(*

.. <legal notes>

legal notes
=================
| SPDX-FileCopyrightText: © 2026 Oleksandr Tiutyk <trofimich@gmail.com>
| SPDX-License-Identifier: LGPL-3.0-only
| For details check: LGPL-3.0-only_

.. _LGPL-3.0-only: https://www.gnu.org/licenses/lgpl-3.0.en.html

.. </legal notes>

*)

FUNCTION_BLOCK ABSTRACT LeafAutomationComponent EXTENDS AutomationComponent IMPLEMENTS IChildAutomationComponent
VAR
	{attribute 'hide'} 
	_Parent : IParentAutomationComponent;
END_VAR

METHOD FINAL BubbleEvent
VAR_INPUT
	event : TOF_Core.IEvent;
END_VAR
VAR
	stopPropagation : BOOL;
	
	parentAsBubbleEventDispatcher : TOF_Core.IBubbleEventDispatcher;
END_VAR
OnEventReceived(event := event, stopPropagation => stopPropagation);

IF stopPropagation THEN
	RETURN;
END_IF

IF __QUERYINTERFACE(Parent, parentAsBubbleEventDispatcher) THEN
	parentAsBubbleEventDispatcher.BubbleEvent(event);
END_IF
END_METHOD

METHOD FINAL Disable
VAR
	i : TOF_Core.INT_INDEX;
	
	child : IChildAutomationComponent;
END_VAR
VAR_INST
	disabling : BOOL;
END_VAR
IF NOT _Enabled OR_ELSE disabling THEN
	RETURN;
END_IF

disabling := TRUE;

__TRY
	OnDisable();
	
	_Enabled := FALSE;
	
	disabling := FALSE;	
__CATCH		
	disabling := FALSE;
	
	TOF_Core.ExceptionManager.ReThrowLastException();
__ENDTRY
END_METHOD

METHOD FINAL Enable
VAR_INPUT
	includeChildren : BOOL := TRUE;
END_VAR
VAR
	i : TOF_Core.INT_INDEX;
	
	child : IChildAutomationComponent;

	exceptionCode : __SYSTEM.ExceptionCode;
	exception : TOF_Core.IException;	
END_VAR
VAR_INST
	enabling : BOOL;
END_VAR
IF _Enabled OR_ELSE enabling THEN
	RETURN;
END_IF

enabling := TRUE;

__TRY
	OnEnable();
	
	IF _Parent <> 0 AND_THEN NOT _Parent.Enabled THEN
		_Parent.Enable(FALSE);
	END_IF
	
	_Enabled := TRUE;
	
	enabling := FALSE;
__CATCH		
	enabling := FALSE;
	
	TOF_Core.ExceptionManager.ReThrowLastException();
__ENDTRY
END_METHOD

METHOD FINAL Execute
VAR
	inputDevice : IInputDevice;	
	outputDevice : IOutputDevice;	

	exceptionCode : __SYSTEM.ExceptionCode;
	exception : TOF_Core.IException;	
	exceptionReaction : TOF_Core.EXCEPTION_REACTION;
END_VAR
IF NOT Enabled OR_ELSE (_OperationalState <> OPERATIONAL_STATE.WORKING AND_THEN _OperationalState <> OPERATIONAL_STATE.STOPPED) THEN
	RETURN;
END_IF

IF __QUERYINTERFACE(THIS^, inputDevice) THEN
	inputDevice.ProcessInput();
END_IF

CASE _OperationalState OF
	OPERATIONAL_STATE.WORKING:
		// automatic non-critical error recovering
		IF _OperationalState = OPERATIONAL_STATE.WORKING AND_THEN HasError AND_THEN _Error.Severity <> TOF_Core.ERROR_SEVERITY.CRITICAL THEN
			_Error.Clear();
			
			__TRY
				OnRecover();
			__CATCH(exceptionCode)		
				exception := TOF_Core.ExceptionManager.GetLastException(exceptionCode);
								
				exceptionReaction := OnHandleException(exception, 'OnRecover');
			
				ProcessException(exception, exceptionReaction, "OnRecover error");
			
				IF exceptionReaction = TOF_Core.EXCEPTION_REACTION.SET_ERROR_AND_STOP THEN
					RETURN;
				END_IF		
			__ENDTRY
		END_IF
		
		__TRY
			OnWorking();
		__CATCH(exceptionCode)
			exception := TOF_Core.ExceptionManager.GetLastException(exceptionCode);	
		
			exceptionReaction := OnHandleException(exception, 'OnWorking');
		
			ProcessException(exception, exceptionReaction, "OnBeforeChildrenWorking error");
		
			IF exceptionReaction = TOF_Core.EXCEPTION_REACTION.SET_ERROR_AND_STOP THEN
				RETURN;		
			END_IF
		__ENDTRY
		
	OPERATIONAL_STATE.STOPPED:
		__TRY
			OnStopped();
		__CATCH(exceptionCode)
			exception := TOF_Core.ExceptionManager.GetLastException(exceptionCode);	
		
			exceptionReaction := OnHandleException(exception, 'OnStopped');
		
			TOF_Core.LogManager.TryLogException(exception, GetErrorSeverityByExceptionReaction(exceptionReaction), "AutomationComponent", "AutomationComponent.OnStopped");
		__ENDTRY	
END_CASE

IF __QUERYINTERFACE(THIS^, outputDevice) THEN
	outputDevice.ProcessOutput();
END_IF
END_METHOD

METHOD FB_init : BOOL
VAR_INPUT
	(* if TRUE, the retain variables are initialized (warm start / cold start)*)
	bInitRetains	: BOOL;
	(* if TRUE, the instance afterwards gets moved into the copy code (online change)*)
	bInCopyCode	: BOOL;
	name : WSTRING;
	parent : IParentAutomationComponent;
END_VAR
_Parent := parent;
END_METHOD

METHOD FINAL Initialize : BOOL
VAR
	i : TOF_Core.INT_INDEX;
	
	thisAsParentComponent : IChildAutomationComponent;
	parent : IAutomationComponent;
	child : IChildAutomationComponent;
	
	exceptionCode : __SYSTEM.ExceptionCode;
	exception : TOF_Core.IException;
	
	initializationTimeoutException : TOF_Core.TimeoutException;
	notSpecifiedException : TOF_Core.DataMemberNotSpecifiedException;
END_VAR
IF _OperationalState <> OPERATIONAL_STATE.INITIALIZING THEN
	Initialize := _OperationalState <> OPERATIONAL_STATE.INVALID;
	
	RETURN;
END_IF

__TRY
	_InitializationTimer(IN := TRUE, PT := Parameters.InitializationTimeout);
	
	IF _InitializationTimer.Q THEN		
		initializationTimeoutException.ThrowByObject(THIS^, __POUNAME(), __POSITION(), _InitializationTimer.PT, TOF_Core.WideStrings.Concat255("Initialization timeout ", TO_WSTRING(_InitializationTimer.PT), " elapsed"));
	END_IF
	
	IF __QUERYINTERFACE(THIS^, thisAsParentComponent) AND_THEN (parent := thisAsParentComponent.Parent) = 0 THEN
		notSpecifiedException.ThrowByObject(THIS^, __POUNAME(), __POSITION(), 'Parent');						
	END_IF

	Initialize := OnInitializing();
	
	IF Initialize THEN
		SetOperationalState(OPERATIONAL_STATE.WORKING, "Successfull initialization");
	END_IF	
__CATCH(exceptionCode)
	exception := TOF_Core.ExceptionManager.GetLastException(exceptionCode);
	
	ProcessException(exception, TOF_Core.EXCEPTION_REACTION.SET_ERROR_AND_CONTINUE, "Initialization error");					
__ENDTRY
END_METHOD

METHOD PROTECTED OnDisable
END_METHOD

METHOD PROTECTED OnEnable
END_METHOD

METHOD PROTECTED OnInitializing : BOOL
OnInitializing := TRUE;
END_METHOD

METHOD PROTECTED OnReset
END_METHOD

METHOD PROTECTED OnStopped
END_METHOD

METHOD PROTECTED OnWorking
END_METHOD

{attribute 'monitoring' := 'call'}
PROPERTY FINAL Parent : IParentAutomationComponent
GET
Parent := _Parent;
END_GET
END_PROPERTY

METHOD FINAL Reset
VAR
	exceptionCode : __SYSTEM.ExceptionCode;
	exception : TOF_Core.IException;	
	exceptionReaction : TOF_Core.EXCEPTION_REACTION;
	
	i : TOF_Core.INT_INDEX;
		
	child : IChildAutomationComponent;	
END_VAR
IF NOT Enabled OR_ELSE _OperationalState <> OPERATIONAL_STATE.STOPPED THEN
	RETURN;
END_IF

_Error.Clear();

__TRY
	OnReset();
__CATCH(exceptionCode)		
	exception := TOF_Core.ExceptionManager.GetLastException(exceptionCode);
					
	exceptionReaction := OnHandleException(exception, 'OnReset');

	ProcessException(exception, exceptionReaction, "OnReset error");

	IF exceptionReaction = TOF_Core.EXCEPTION_REACTION.SET_ERROR_AND_STOP THEN
		RETURN;
	END_IF
__ENDTRY
END_METHOD

METHOD FINAL Stop
VAR_INPUT
	reason : WSTRING(255) := "External stop";
END_VAR
VAR
	exceptionCode : __SYSTEM.ExceptionCode;
	exception : TOF_Core.IException;	

	i : TOF_Core.INT_INDEX;
	
	child : IChildAutomationComponent;
END_VAR
IF NOT _Enabled OR_ELSE _OperationalState <> OPERATIONAL_STATE.WORKING THEN
	RETURN;
END_IF

SetOperationalState(OPERATIONAL_STATE.STOPPED, reason);
END_METHOD

END_FUNCTION_BLOCK

(* stored: Version 1.1.0.1
   POU LeafAutomationComponent: Id {7c21300f-1ad4-4217-9d49-d0f060249ecb}, SpecialFunc None
   Folder Methods to override: Id {ca4cde0e-9a44-45fe-a0e4-7b7ca4e0c8a7}
   Method BubbleEvent: Id {42cce6a6-4219-41f5-a23e-d08f59aa4482}
   Method Disable: Id {e7be34cc-e7d9-4568-8b6a-522ee606d568}
   Method Enable: Id {f7b45f9a-e580-4c1c-b27c-81b9ee1ab687}
   Method Execute: Id {54d74276-cad2-4fd8-8917-0010f6191e07}
   Method FB_init: Id {3ffe21cc-32bd-4767-9934-eaac8121d03b}
   Method Initialize: Id {3f657450-0a0b-4d21-8c85-c39655b515b8}
   Method OnDisable: Id {da5e244e-35a1-47cd-8144-7c7c3577035d}
   Method OnEnable: Id {7ab79cf0-ed24-4ab4-b074-f58d9b879980}
   Method OnInitializing: Id {87d0edb2-3f9d-4cdc-be5a-51ee4854c5ea}
   Method OnReset: Id {1437f653-2dca-4516-a643-9a7052ba8f91}
   Method OnStopped: Id {38cbad82-8eb7-4619-bb79-98729012ae5d}
   Method OnWorking: Id {02692fef-98a0-451c-b7a8-b233e155c1c5}
   Property Parent: Id {8fb3d4d7-c400-4c92-9c99-1346029f28e7}
   Get Get: Id {91af78c8-f2e0-4384-ac9d-b26f89ba6059}
   Method Reset: Id {39108ecc-e8fc-41d2-84a8-8d829dba9e49}
   Method Stop: Id {73828ae5-99ee-4c51-a656-702f6c6b2044} *)
